FUNCTION_BLOCK FB_Max_Value_Test EXTENDS TcUnit.FB_TestSuite
VAR
END_VAR

FirstValueIsBiggest();
SecondValueIsBiggest();
ValuesAreEqual();

METHOD FirstValueIsBiggest
VAR
	Maximum : FB_Max_Value;
	Result: LREAL;
	ExpectedMax : LREAL := 3;
END_VAR
TEST('TEST: First Value Is Biggest');

Maximum(value1 := 3, value2 := 1, result => Result);

AssertEquals(Expected := ExpectedMax,
			Actual := Result,
			Message := 'Max value not found');

TEST_FINISHED();
END_METHOD

METHOD SecondValueIsBiggest
VAR
	Maximum : FB_Max_Value;
	Result : LREAL;
	ExpectedMax : LREAL := 9;
	
END_VAR
TEST('TEST: Second value is largest');

Maximum(value1 := 1, value2 := 9, result => Result);

AssertEquals(Expected := ExpectedMax,
			Actual := Result,
			Message := 'Largest value not found');

TEST_FINISHED();
END_METHOD

METHOD ValuesAreEqual
VAR
	Maximum : FB_Max_Value;
	Result : LREAL;
	ExpectedMax : LREAL := -999;
END_VAR
TEST('Checks output if both input values are the same');

Maximum(value1 := -999,
		value2 := -999,
		result => Result);

AssertEquals(Expected := ExpectedMax,
			Actual := Result,
			Message := 'Largest value not found');
			
TEST_FINISHED();
END_METHOD

END_FUNCTION_BLOCK

(* stored: Version 1.1.0.1, ProductVersion 3.1.4024.13
   POU FB_Max_Value_Test: Id {adf3ba5e-5a03-434b-a82b-cde5610e43c9}, SpecialFunc None
   Method FirstValueIsBiggest: Id {b97959e4-bdbd-4f26-b6cb-1adfe065b1c9}
   Method SecondValueIsBiggest: Id {91cb6d46-0c42-490b-8e47-19d341bcf3b0}
   Method ValuesAreEqual: Id {7319594c-6dd5-4b37-80e4-5e5eb5741678} *)
